// TIA Portal project "Sortier_Station_1" (V20)

(* hardware
DEVICE "S7-1500/ET200MP-Station_1"  S7-1500 station
   slot 0: "Profilschiene_0"  Rack  6ES7 590-1***0-0AA0
   slot 1: "PLC_1"  CPU 1513-1 PN  6ES7 513-1AM03-0AB0  V4.0
      slot 3: "CPU-Display_1"  6ES7591-1AA00-0AA0
      slot 32768: "PROFINET-Schnittstelle_1"  X1
         slot 32769: "Port_1"  X1 P1
         slot 32770: "Port_2"  X1 P2
      slot 34817: "Virtual CP interface port_1"  Virtual CP interface port  Virtual CP interface port FW V4.0
   slot 2: "DI 16x24VDC BA_1"  DI 16x24VDC BA  6ES7 521-1BH10-0AA0  V1.1
   slot 3: "DQ 16x24VDC/0.5A ST_1"  DQ 16x24VDC/0.5A ST  6ES7 522-1BH00-0AB0  V2.0
   slot 4: "AI 8xU/I/R/RTD BA_1"  AI 8xU/I/R/RTD BA  6ES7 531-7QF00-0AB0  V1.0
   slot 5: "AQ 8xU/I HS_1"  AQ 8xU/I HS  6ES7 532-5HF00-0AB0  V2.2
   slot 6: "AI 8xU/I/R/RTD BA_2"  AI 8xU/I/R/RTD BA  6ES7 531-7QF00-0AB0  V1.0
   slot 7: "AQ 8xU/I HS_2"  AQ 8xU/I HS  6ES7 532-5HF00-0AB0  V2.2
*)

// ===== PLC "PLC_1"  CPU 1513-1 PN =====

VAR_GLOBAL   // PLC tag table "Standard-Variablentabelle"
   "PlcLabConnectIn01" AT %ID32760 : DWord;
   "PlcLabConnectIn02" AT %ID32764 : DWord;
   "PlcLabConnectOut01" AT %QD32760 : DWord;
   "PlcLabConnectOut02" AT %QD32764 : DWord;
   "Clock_Byte" AT %MB0 : Byte;
   "Clock_10Hz" AT %M0.0 : Bool;
   "Clock_5Hz" AT %M0.1 : Bool;
   "Clock_2.5Hz" AT %M0.2 : Bool;
   "Clock_2Hz" AT %M0.3 : Bool;
   "Clock_1.25Hz" AT %M0.4 : Bool;
   "Clock_1Hz" AT %M0.5 : Bool;
   "Clock_0.625Hz" AT %M0.6 : Bool;
   "Clock_0.5Hz" AT %M0.7 : Bool;
END_VAR

VAR_GLOBAL   // PLC tag table "Eingaenge"
   "S1" AT %I0.0 : Bool;   // Not-Aus Schalter
   "S2" AT %I0.1 : Bool;   // Betriebsschalter
   "S3" AT %I0.2 : Bool;   // Starttaster
   "S4" AT %I0.3 : Bool;   // Stopptaster
   "S5" AT %I0.4 : Bool;   // Resettaster
   "6b1" AT %I1.0 : Bool;   // Lichttaster Auslauf (Sortierer rechts)
   "1b1" AT %ID30 : DInt;   // Visionsensor am Eingang
   "4b1" AT %E0.6 : Bool;   // Lichttaster nach Sortierer rechts
   "5b1" AT %E0.7 : Bool;   // Lichttaster nach Sortierer mitte
   "6b2" AT %E1.1 : Bool;   // Lichttaster Auslauf (Sortierer mitte)
   "6b3" AT %E1.2 : Bool;   // Lichttaster Auslauf (Sortierer links)
   "3b1" AT %E0.5 : Bool;   // Lichttaster vor Sortierer rechts
END_VAR

VAR_GLOBAL   // PLC tag table "Ausgaenge"
   "H1" AT %Q0.2 : Bool;   // Startleuchte
   "H2" AT %Q0.3 : Bool;   // Stoppleuchte
   "H3" AT %Q0.4 : Bool;   // Resetleuchte
   "M1" AT %A0.5 : Bool;   // Zulauf Förderband
   "M2" AT %A0.6 : Bool;   // Auslauf Förderband
   "M3" AT %A0.7 : Bool;   // Stopp-Barriere
   "4M1" AT %Q1.3 : Bool;   // Sortierer (rechts)
   "5M1" AT %Q1.4 : Bool;   // Sortierer (mittig)
   "6M1" AT %Q1.5 : Bool;   // Sortierer (links)
   "D1" AT %QD30 : DInt;   // Zähleranzeige (rechts)
   "D2" AT %QD34 : DInt;   // Zähleranzeige (mittig)
   "D3" AT %QD38 : DInt;   // Zähleranzeige (links)
   "4M2" AT %A1.0 : Bool;   // Sortiererband (rechts)
   "5M2" AT %A1.1 : Bool;   // Sortiererband (mittig)
   "6M2" AT %A1.2 : Bool;   // Sortiererband (links)
END_VAR

DATA_BLOCK "Zaehlerdaten"   // DB1
{ S7_Optimized_Access := 'TRUE' }
VERSION : 0.1
// stored: InstanceOfName Zaehlersteuerung
"Zaehlersteuerung"
BEGIN
END_DATA_BLOCK

DATA_BLOCK "Sortierdaten"   // DB2
{ S7_Optimized_Access := 'TRUE' }
VERSION : 0.1
   VAR
      Anlagendaten : Struct
         NotAus_aktiv : Bool;
         NotAus_angeschaltet : Bool;
         Anlage_aktiv : Bool;
         Anlage_angeschaltet : Bool;
      END_STRUCT;
      Betriebsdaten : Struct
         Teil_erkannt : Struct
            Blau : Bool;
            Gruen : Bool;
            Grau : Bool;
         END_STRUCT;
         NTRIG_3b1 : Bool;
         PTRIG_4b1 : Bool;
         PTRIG_5b1 : Bool;
         Teil_raus : Struct
            Blau : Bool;
            Gruen : Bool;
            Grau : Bool;
         END_STRUCT;
         Iterator_Bauteile : USInt;
         Bauteile : Array[0..4] of USInt;   // Eine Warteschlange, um das erste Bauteil zu bestimmen
         Auslauf_Positionen : Array[0..2] of USInt;   // Die aktuelle Position eines Bauteils auf dem Auslassband
         Sortierermotoren : Struct
            "1M1" : Bool;
            "2M1" : Bool;
            "3M1" : Bool;
         END_STRUCT;
      END_STRUCT;
      Fehler : Struct
         Stack_verschieben : Int;
      END_STRUCT;
   END_VAR
BEGIN
END_DATA_BLOCK

FUNCTION_BLOCK "Zaehlersteuerung"   // FB1, FBD
{ S7_Optimized_Access := 'TRUE' }
VERSION : 0.1
   VAR
      Bauteil_Zaehler_Blau : "Bauteil_Zaehler";
      Bauteil_Zaehler_Gruen : "Bauteil_Zaehler";
      Bauteil_Zaehler_Grau : "Bauteil_Zaehler";
   END_VAR
   VAR CONSTANT
      Blaues_Bauteil : Int := 1;
      Gruenes_Bauteil : Int := 2;
      Graues_Bauteil : Int := 3;
   END_VAR
BEGIN

REGION Network 1: Zähler (blaue Teile)
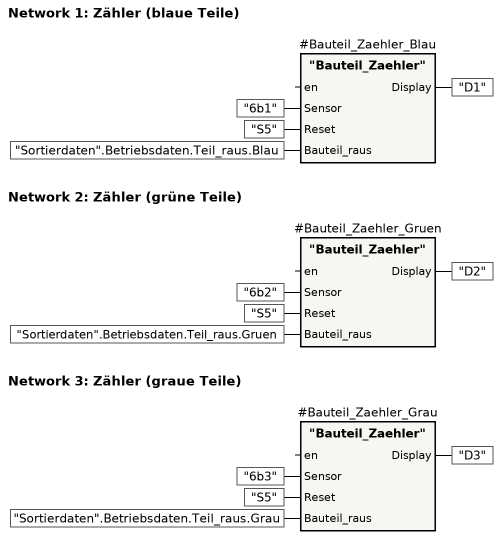
   #Bauteil_Zaehler_Blau(Sensor := "6b1",   // "Bauteil_Zaehler"
                         Reset := "S5",
                         Bauteil_raus := "Sortierdaten".Betriebsdaten.Teil_raus.Blau,
                         Display => "D1");
END_REGION

REGION Network 2: Zähler (grüne Teile)
   #Bauteil_Zaehler_Gruen(Sensor := "6b2",   // "Bauteil_Zaehler"
                          Reset := "S5",
                          Bauteil_raus := "Sortierdaten".Betriebsdaten.Teil_raus.Gruen,
                          Display => "D2");
END_REGION

REGION Network 3: Zähler (graue Teile)
   #Bauteil_Zaehler_Grau(Sensor := "6b3",   // "Bauteil_Zaehler"
                         Reset := "S5",
                         Bauteil_raus := "Sortierdaten".Betriebsdaten.Teil_raus.Grau,
                         Display => "D3");
END_REGION
END_FUNCTION_BLOCK

FUNCTION_BLOCK "Bauteil_Zaehler"   // FB2, FBD
{ S7_Optimized_Access := 'TRUE' }
VERSION : 0.1
   VAR_INPUT
      Sensor : Bool;
      Reset : Bool;
   END_VAR
   VAR_OUTPUT
      Display : DInt;
   END_VAR
   VAR_IN_OUT
      Bauteil_raus : Bool;
   END_VAR
   VAR RETAIN
      IEC_Zaehler_Bauteil_Farbe : CTU_INT;
   END_VAR
   VAR
      Anzahl : Int;
      NTRIG_Sensor : Bool;
   END_VAR
   VAR_TEMP   // added for the SCL form of the ladder/FBD networks
      _w1 : Bool;
   END_VAR
BEGIN

REGION Network 1
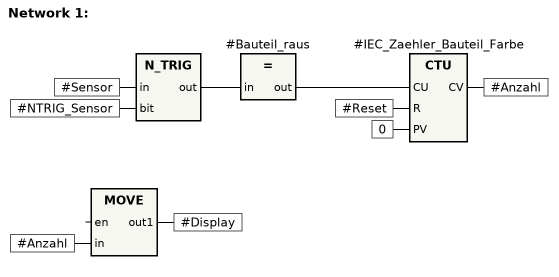
   #_w1 := NOT #Sensor AND #NTRIG_Sensor;   // falling edge
   #NTRIG_Sensor := #Sensor;
   #Bauteil_raus := #_w1;
   #IEC_Zaehler_Bauteil_Farbe(CU := #_w1, R := #Reset, PV := 0, CV => #Anzahl);   // CTU
   #Display := #Anzahl;
END_REGION
END_FUNCTION_BLOCK

FUNCTION "Bandsteuerung" : Void   // FC1, FBD
{ S7_Optimized_Access := 'TRUE' }
VERSION : 0.1
BEGIN

REGION Network 1: Bandsteuerung
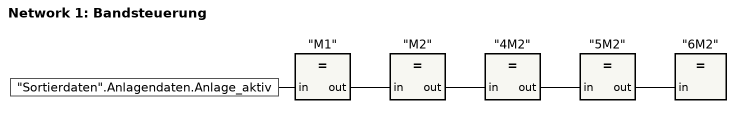
   "M1" := "Sortierdaten".Anlagendaten.Anlage_aktiv;
   "M2" := "Sortierdaten".Anlagendaten.Anlage_aktiv;
   "4M2" := "Sortierdaten".Anlagendaten.Anlage_aktiv;
   "5M2" := "Sortierdaten".Anlagendaten.Anlage_aktiv;
   "6M2" := "Sortierdaten".Anlagendaten.Anlage_aktiv;
END_REGION
END_FUNCTION

FUNCTION "Sortiersteuerung" : Void   // FC2, FBD
{ S7_Optimized_Access := 'TRUE' }
VERSION : 0.1
   VAR CONSTANT
      Blaues_Bauteil : USInt := 1;
      Gruenes_Bauteil : USInt := 2;
      Graues_Bauteil : USInt := 3;
      Bauteile_Max : USInt := 4;
   END_VAR
   VAR_TEMP   // added for the SCL form of the ladder/FBD networks
      _w1 : Bool;
      _w2 : Bool;
      _w3 : Bool;
   END_VAR
BEGIN

REGION Network 1: Iterator zurücksetzen
   // Falls es Probleme gibt mit der Software (z.B. Iterator wird -1 oder gößer 10) kann das Array nicht genutzt werden. Deshalb soll wenn die Anlage aus ist, der Iterator zurückgesetzt werden.
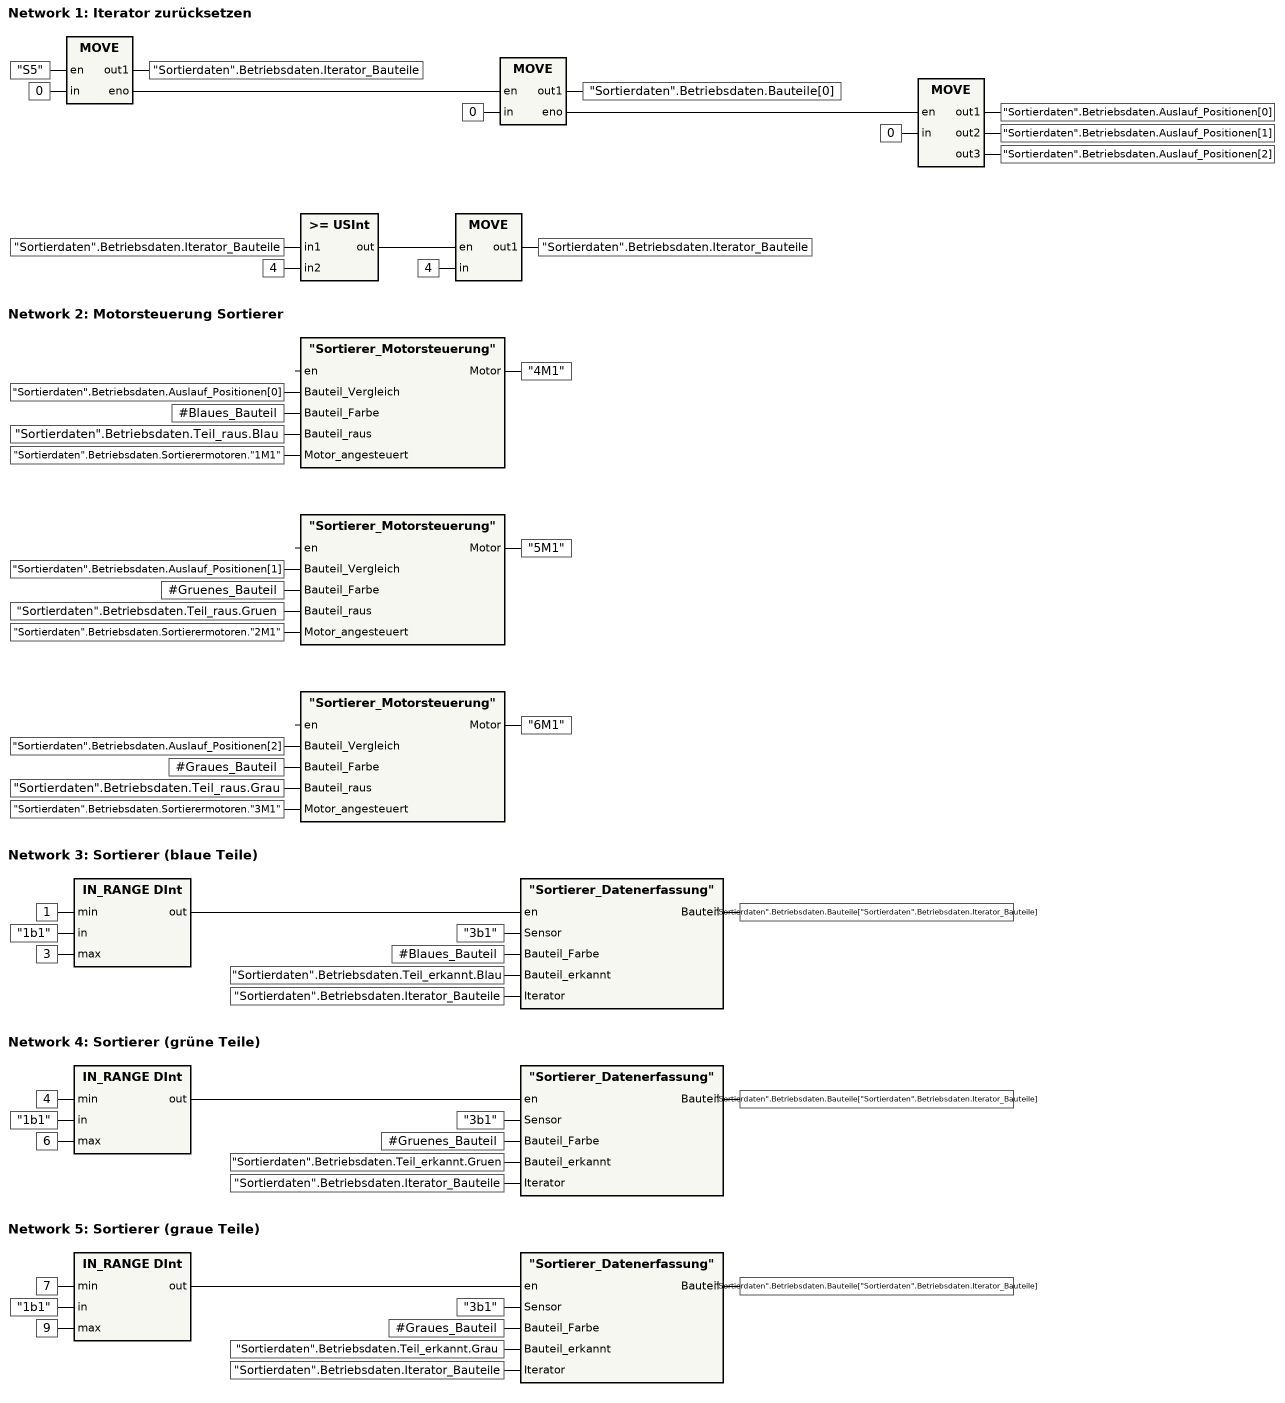
   IF "S5" THEN
       "Sortierdaten".Betriebsdaten.Iterator_Bauteile := 0;
       "Sortierdaten".Betriebsdaten.Bauteile[0] := 0;
       "Sortierdaten".Betriebsdaten.Auslauf_Positionen[0] := 0;
       "Sortierdaten".Betriebsdaten.Auslauf_Positionen[1] := 0;
       "Sortierdaten".Betriebsdaten.Auslauf_Positionen[2] := 0;
   END_IF;
   IF "Sortierdaten".Betriebsdaten.Iterator_Bauteile >= 4 THEN
       "Sortierdaten".Betriebsdaten.Iterator_Bauteile := 4;
   END_IF;
END_REGION

REGION Network 2: Motorsteuerung Sortierer
   "Sortierer_Motorsteuerung"(Bauteil_Vergleich := "Sortierdaten".Betriebsdaten.Auslauf_Positionen[0],
                           Bauteil_Farbe := #Blaues_Bauteil,
                           Bauteil_raus := "Sortierdaten".Betriebsdaten.Teil_raus.Blau,
                           Motor_angesteuert := "Sortierdaten".Betriebsdaten.Sortierermotoren."1M1",
                           Motor => "4M1");
   "Sortierer_Motorsteuerung"(Bauteil_Vergleich := "Sortierdaten".Betriebsdaten.Auslauf_Positionen[1],
                           Bauteil_Farbe := #Gruenes_Bauteil,
                           Bauteil_raus := "Sortierdaten".Betriebsdaten.Teil_raus.Gruen,
                           Motor_angesteuert := "Sortierdaten".Betriebsdaten.Sortierermotoren."2M1",
                           Motor => "5M1");
   "Sortierer_Motorsteuerung"(Bauteil_Vergleich := "Sortierdaten".Betriebsdaten.Auslauf_Positionen[2],
                           Bauteil_Farbe := #Graues_Bauteil,
                           Bauteil_raus := "Sortierdaten".Betriebsdaten.Teil_raus.Grau,
                           Motor_angesteuert := "Sortierdaten".Betriebsdaten.Sortierermotoren."3M1",
                           Motor => "6M1");
END_REGION

REGION Network 3: Sortierer (blaue Teile)
   IF (1 <= "1b1") AND ("1b1" <= 3) THEN
       "Sortierer_Datenerfassung"(Sensor := "3b1",
                               Bauteil_Farbe := #Blaues_Bauteil,
                               Bauteil_erkannt := "Sortierdaten".Betriebsdaten.Teil_erkannt.Blau,
                               Iterator := "Sortierdaten".Betriebsdaten.Iterator_Bauteile,
                               Bauteil => "Sortierdaten".Betriebsdaten.Bauteile["Sortierdaten".Betriebsdaten.Iterator_Bauteile]);
   END_IF;
END_REGION

REGION Network 4: Sortierer (grüne Teile)
   IF (4 <= "1b1") AND ("1b1" <= 6) THEN
       "Sortierer_Datenerfassung"(Sensor := "3b1",
                               Bauteil_Farbe := #Gruenes_Bauteil,
                               Bauteil_erkannt := "Sortierdaten".Betriebsdaten.Teil_erkannt.Gruen,
                               Iterator := "Sortierdaten".Betriebsdaten.Iterator_Bauteile,
                               Bauteil => "Sortierdaten".Betriebsdaten.Bauteile["Sortierdaten".Betriebsdaten.Iterator_Bauteile]);
   END_IF;
END_REGION

REGION Network 5: Sortierer (graue Teile)
   IF (7 <= "1b1") AND ("1b1" <= 9) THEN
       "Sortierer_Datenerfassung"(Sensor := "3b1",
                               Bauteil_Farbe := #Graues_Bauteil,
                               Bauteil_erkannt := "Sortierdaten".Betriebsdaten.Teil_erkannt.Grau,
                               Iterator := "Sortierdaten".Betriebsdaten.Iterator_Bauteile,
                               Bauteil => "Sortierdaten".Betriebsdaten.Bauteile["Sortierdaten".Betriebsdaten.Iterator_Bauteile]);
   END_IF;
END_REGION

REGION Network 6: Arraysteuerung (Einlass)
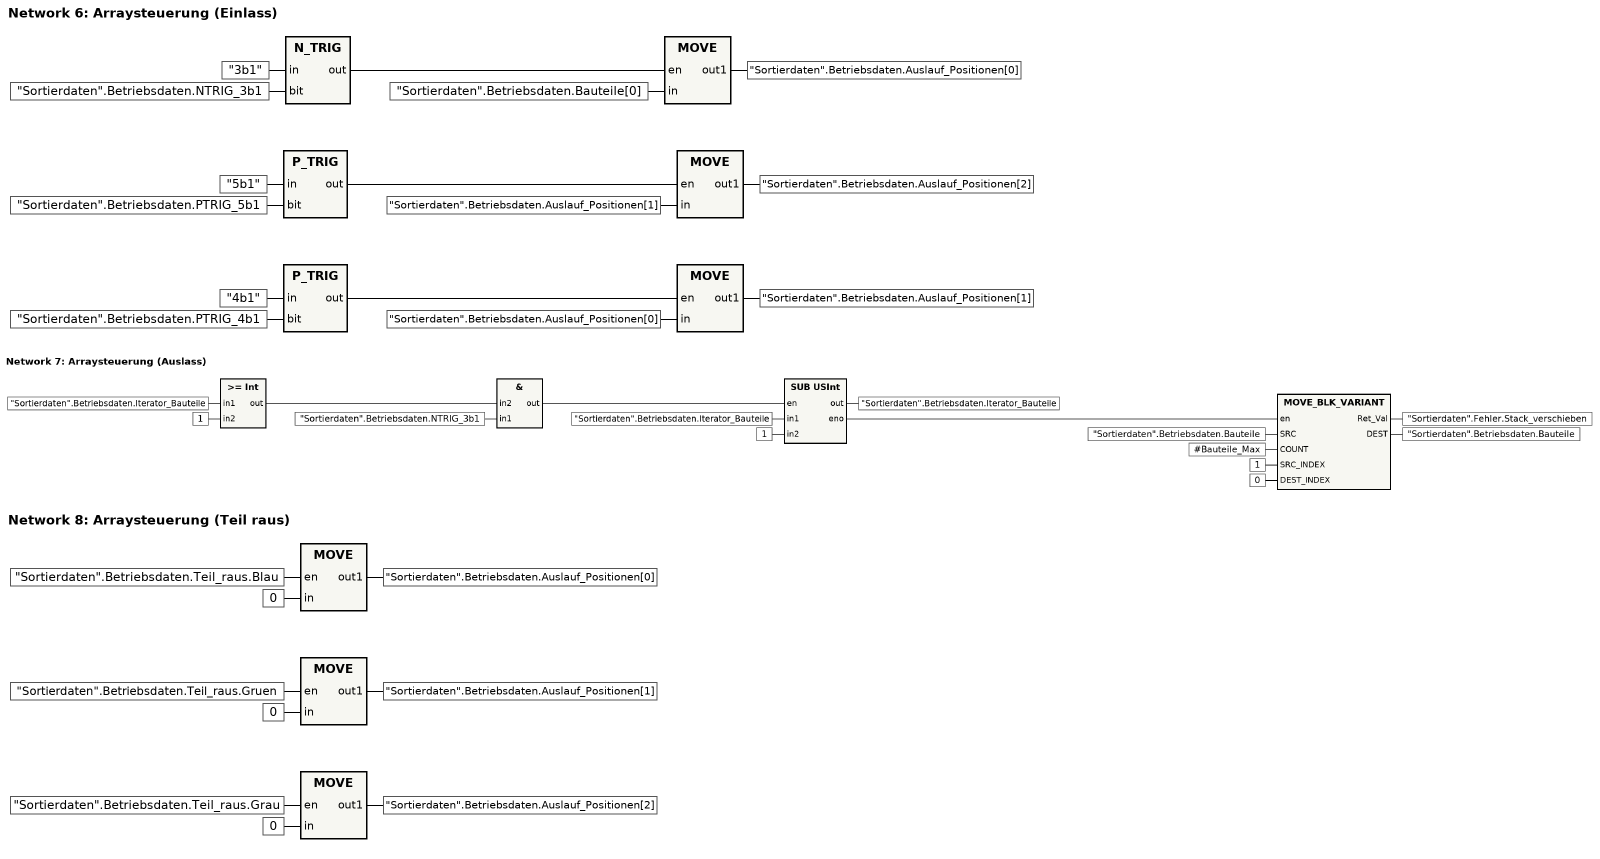
   #_w1 := NOT "3b1" AND "Sortierdaten".Betriebsdaten.NTRIG_3b1;   // falling edge
   "Sortierdaten".Betriebsdaten.NTRIG_3b1 := "3b1";
   IF #_w1 THEN
       "Sortierdaten".Betriebsdaten.Auslauf_Positionen[0] := "Sortierdaten".Betriebsdaten.Bauteile[0];
   END_IF;
   #_w2 := "5b1" AND NOT "Sortierdaten".Betriebsdaten.PTRIG_5b1;   // rising edge
   "Sortierdaten".Betriebsdaten.PTRIG_5b1 := "5b1";
   IF #_w2 THEN
       "Sortierdaten".Betriebsdaten.Auslauf_Positionen[2] := "Sortierdaten".Betriebsdaten.Auslauf_Positionen[1];
   END_IF;
   #_w3 := "4b1" AND NOT "Sortierdaten".Betriebsdaten.PTRIG_4b1;   // rising edge
   "Sortierdaten".Betriebsdaten.PTRIG_4b1 := "4b1";
   IF #_w3 THEN
       "Sortierdaten".Betriebsdaten.Auslauf_Positionen[1] := "Sortierdaten".Betriebsdaten.Auslauf_Positionen[0];
   END_IF;
END_REGION

REGION Network 7: Arraysteuerung (Auslass)
   #_w1 := ("Sortierdaten".Betriebsdaten.Iterator_Bauteile >= 1) AND "Sortierdaten".Betriebsdaten.NTRIG_3b1;
   IF #_w1 THEN
       "Sortierdaten".Betriebsdaten.Iterator_Bauteile := "Sortierdaten".Betriebsdaten.Iterator_Bauteile - 1;
       "Sortierdaten".Fehler.Stack_verschieben := MOVE_BLK_VARIANT(SRC := "Sortierdaten".Betriebsdaten.Bauteile,
                               COUNT := #Bauteile_Max,
                               SRC_INDEX := 1,
                               DEST_INDEX := 0,
                               DEST => "Sortierdaten".Betriebsdaten.Bauteile);
   END_IF;
END_REGION

REGION Network 8: Arraysteuerung (Teil raus)
   IF "Sortierdaten".Betriebsdaten.Teil_raus.Blau THEN
       "Sortierdaten".Betriebsdaten.Auslauf_Positionen[0] := 0;
   END_IF;
   IF "Sortierdaten".Betriebsdaten.Teil_raus.Gruen THEN
       "Sortierdaten".Betriebsdaten.Auslauf_Positionen[1] := 0;
   END_IF;
   IF "Sortierdaten".Betriebsdaten.Teil_raus.Grau THEN
       "Sortierdaten".Betriebsdaten.Auslauf_Positionen[2] := 0;
   END_IF;
END_REGION
END_FUNCTION

FUNCTION "Anlagensteuerung" : Void   // FC4, FBD
{ S7_Optimized_Access := 'TRUE' }
VERSION : 0.1
   VAR_INPUT
      "Not-Aus" : Bool;
      "Betrieb-ein" : Bool;
      Start : Bool;
      Stopp : Bool;
      Reset : Bool;
   END_VAR
   VAR_OUTPUT
      NotAus_ein : Bool;
      Anlage_ein : Bool;
   END_VAR
   VAR_IN_OUT
      NotAus_aktiv : Bool;
      Anlage_aktiv : Bool;
   END_VAR
BEGIN

REGION Network 1: Anlagensteuerung
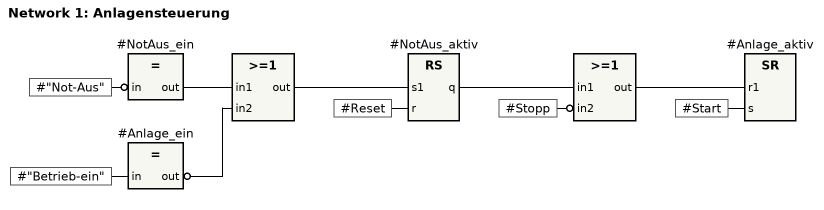
   #NotAus_ein := NOT #"Not-Aus";
   #Anlage_ein := #"Betrieb-ein";
   IF #Reset THEN
       #NotAus_aktiv := FALSE;   // RS flip-flop
   END_IF;
   IF NOT #"Not-Aus" OR NOT #"Betrieb-ein" THEN #NotAus_aktiv := TRUE; END_IF;
   IF #Start THEN
       #Anlage_aktiv := TRUE;   // SR flip-flop
   END_IF;
   IF #NotAus_aktiv OR NOT #Stopp THEN #Anlage_aktiv := FALSE; END_IF;
END_REGION
END_FUNCTION

FUNCTION "Leuchtensteuerung" : Void   // FC5, FBD
{ S7_Optimized_Access := 'TRUE' }
VERSION : 0.1
   VAR_INPUT
      NotAus_aktiv : Bool;
      NotAus_ein : Bool;
      Anlage_ein : Bool;
      Taktmerker : Bool;
   END_VAR
   VAR_OUTPUT
      Start : Bool;
      Stopp : Bool;
      Reset : Bool;
   END_VAR
BEGIN

REGION Network 1: Leuchtensteuerung
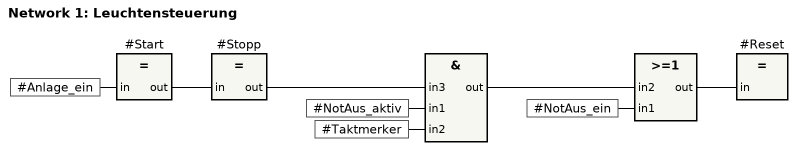
   #Start := #Anlage_ein;
   #Stopp := #Anlage_ein;
   #Reset := (#Anlage_ein AND #NotAus_aktiv AND #Taktmerker) OR #NotAus_ein;
END_REGION
END_FUNCTION

FUNCTION "Sortierer_Motorsteuerung" : Void   // FC6, FBD
{ S7_Optimized_Access := 'TRUE' }
VERSION : 0.1
   VAR_INPUT
      Bauteil_Vergleich : USInt;
      Bauteil_Farbe : USInt;
      Bauteil_raus : Bool;
   END_VAR
   VAR_OUTPUT
      Motor : Bool;
   END_VAR
   VAR_IN_OUT
      Motor_angesteuert : Bool;
   END_VAR
BEGIN

REGION Network 1: Sortierer Motorsteuerung
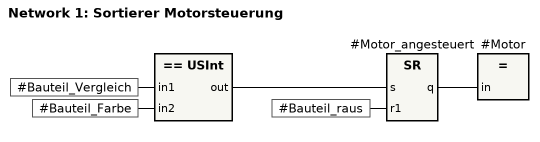
   IF #Bauteil_Vergleich = #Bauteil_Farbe THEN
       #Motor_angesteuert := TRUE;   // SR flip-flop
   END_IF;
   IF #Bauteil_raus THEN #Motor_angesteuert := FALSE; END_IF;
   #Motor := #Motor_angesteuert;
END_REGION
END_FUNCTION

FUNCTION "Sortierer_Datenerfassung" : Void   // FC7, FBD
{ S7_Optimized_Access := 'TRUE' }
VERSION : 0.1
   VAR_INPUT
      Sensor : Bool;
      Bauteil_Farbe : USInt;
   END_VAR
   VAR_OUTPUT
      Bauteil : USInt;
   END_VAR
   VAR_IN_OUT
      Bauteil_erkannt : Bool;
      Iterator : USInt;
   END_VAR
   VAR_TEMP   // added for the SCL form of the ladder/FBD networks
      _w1 : Bool;
      _w2 : Bool;
   END_VAR
BEGIN

REGION Network 1: Sortierer Datenerfassung
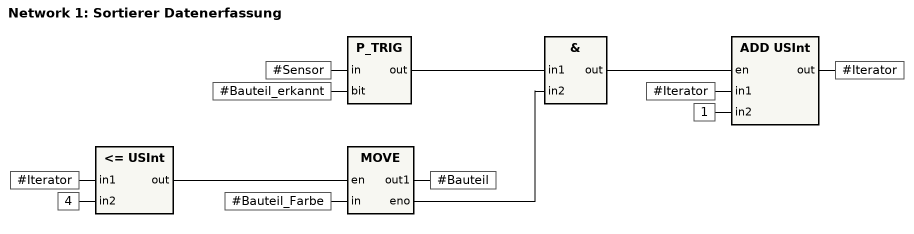
   #_w1 := #Sensor AND NOT #Bauteil_erkannt;   // rising edge
   #Bauteil_erkannt := #Sensor;
   #_w2 := #Iterator <= 4;
   IF #_w2 THEN #Bauteil := #Bauteil_Farbe; END_IF;
   IF #_w1 AND #_w2 THEN #Iterator := #Iterator + 1; END_IF;
END_REGION
END_FUNCTION

ORGANIZATION_BLOCK "Main"   // OB1, FBD, ProgramCycle
TITLE = "Main Program Sweep (Cycle)"
{ S7_Optimized_Access := 'TRUE' }
VERSION : 0.1
   VAR_INPUT
      Initial_Call : Bool;   // Initial call of this OB
      Remanence : Bool;   // =True, if remanent data are available
   END_VAR
BEGIN

REGION Network 1
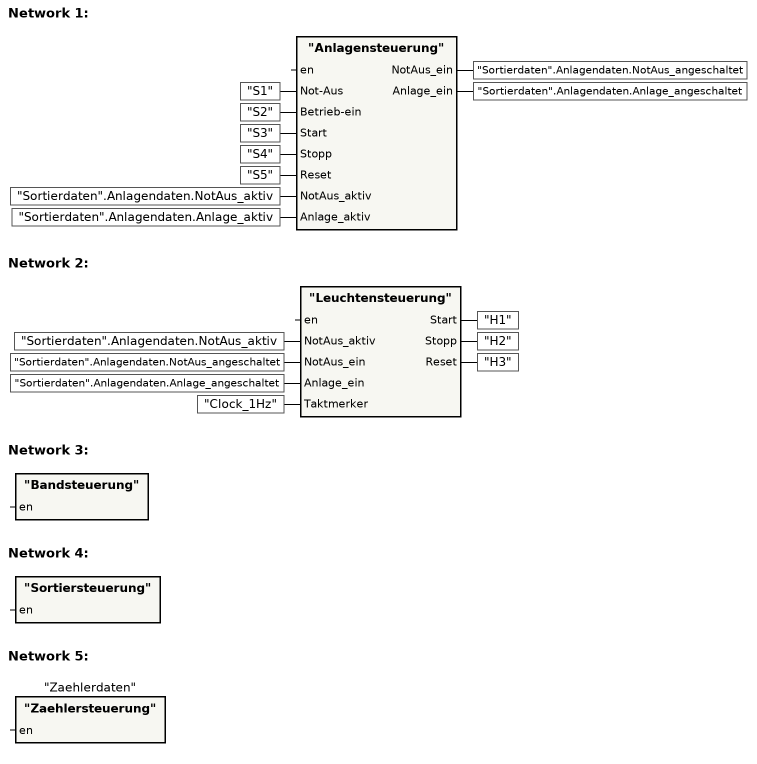
   "Anlagensteuerung"("Not-Aus" := "S1",
                      "Betrieb-ein" := "S2",
                      Start := "S3",
                      Stopp := "S4",
                      Reset := "S5",
                      NotAus_aktiv := "Sortierdaten".Anlagendaten.NotAus_aktiv,
                      Anlage_aktiv := "Sortierdaten".Anlagendaten.Anlage_aktiv,
                      NotAus_ein => "Sortierdaten".Anlagendaten.NotAus_angeschaltet,
                      Anlage_ein => "Sortierdaten".Anlagendaten.Anlage_angeschaltet);
END_REGION

REGION Network 2
   "Leuchtensteuerung"(NotAus_aktiv := "Sortierdaten".Anlagendaten.NotAus_aktiv,
                       NotAus_ein := "Sortierdaten".Anlagendaten.NotAus_angeschaltet,
                       Anlage_ein := "Sortierdaten".Anlagendaten.Anlage_angeschaltet,
                       Taktmerker := "Clock_1Hz",
                       Start => "H1",
                       Stopp => "H2",
                       Reset => "H3");
END_REGION

REGION Network 3
   "Bandsteuerung"();
END_REGION

REGION Network 4
   "Sortiersteuerung"();
END_REGION

REGION Network 5
   "Zaehlerdaten"();   // "Zaehlersteuerung"
END_REGION
END_ORGANIZATION_BLOCK